INTERFACE I_Unwind EXTENDS I_Module, I_TaskResult, I_Resettable, I_Override, I_ContainStatemachine

PROPERTY Recipe : REFERENCE TO ST_UnwindRecipe
GET
END_GET
END_PROPERTY

PROPERTY UnwindAxis : I_Axis_PTP
GET
END_GET
END_PROPERTY

END_INTERFACE

(* stored: Version 1.1.0.1, ProductVersion 3.1.4026.18
   Itf I_Unwind: Id {ec9a7ee6-9040-4ac9-9c55-4e24b124ad09}
   Property Recipe: Id {c1a092a3-e4e2-4904-89df-e1ff57ca5e9e}
   Get Get: Id {ed471d44-1fdb-476d-94f3-b4eeb8b16777}
   Property UnwindAxis: Id {efb7c0fb-8d86-4c3a-a26b-dc8d600abb2b}
   Get Get: Id {9207b0b2-45f9-4b87-9d18-c85e1c95e304} *)
